FUNCTION InfluxAddData_100Hz : BOOL
VAR_IN_OUT
	Data			: ST_DATA;
	DataCollector	: FB_InfluxDataCollector;
END_VAR

// =================== Test
	DataCollector.Addlreal(	'Test64',                                    Data.Gps.Inputs.x);

END_FUNCTION

(* stored: Version 1.1.0.1, ProductVersion 3.1.4022.11
   POU InfluxAddData_100Hz: Id {840c3c73-e0a8-d3c2-797a-bdfdcdede026}, SpecialFunc None *)
